TYPE DS_EventControl :
STRUCT
	bSignalInput 					: BOOL;
	bHoldingDisable 				: BOOL;
	bTest_InvertedInputEn			: BOOL;
	eEventType						: E_EventType;
	iDelayTimeSV					: INT;
	iDelayTimeEV					: INT;
	bEventOutput					: BOOL;
	bEventBuzzerStop				: BOOL;
	
END_STRUCT
END_TYPE

(* stored: Version 1.1.0.1, ProductVersion 3.1.4024.12
   DUT DS_EventControl: Id {16213165-8c4c-4097-a4ac-b9041145cbab} *)
